PROGRAM PRG_GEM
VAR
	
	(*Pressure Control valve  position*)
	VPC_241_Req_Pos: REAL;
	VPC_242_Req_Pos: REAL;
	
	VPC_361_Req_Pos: REAL;
	VPC_362_Req_Pos: REAL;
	
END_VAR

(* GEM 1*)

(*Gauges*)
GEM1_GBA_41(i_rFULL_SCALE := 10.0 (*Torr*));
GEM1_GBA_42(i_rFULL_SCALE := 0.05 (*Torr*));

(* N2 Cut Off Valves *)
GEM1_VVC_40(i_xExtILK_OK:= US_Aperture_Closed AND US_Turbo_Valves_Open AND US_Turbo_Running); 

(*Flow Control Valves*)
GEM1_VPC_41 (i_xExtIlkOK := TRUE, i_rReqPos:= VPC_241_Req_Pos);
GEM1_VPC_42 (i_xExtIlkOK := TRUE, i_rReqPos:= VPC_242_Req_Pos);


(* GEM 2*)

(*Gauges*)
GEM2_GBA_41(i_rFULL_SCALE := 2.0 (*Torr*));
GEM2_GBA_42(i_rFULL_SCALE := 0.05 (*Torr*));
(* N2 Cut Off Valves *)
GEM2_VVC_40(i_xExtILK_OK:= DS_Aperture_Closed AND DS_Turbo_Valves_Open AND DS_Turbo_Running); 


(*Flow Control Valves*)
GEM2_VPC_41(i_xExtIlkOK := TRUE, i_rReqPos:= VPC_361_Req_Pos);
GEM2_VPC_42(i_xExtIlkOK := TRUE, i_rReqPos:= VPC_362_Req_Pos);

(*Control Loop to be implemented*)

END_PROGRAM

(* stored: Version 1.1.0.1, ProductVersion 3.1.4022.16
   POU PRG_GEM: Id {7151a316-9a63-4501-9ce1-47c00a15e083}, SpecialFunc None *)
